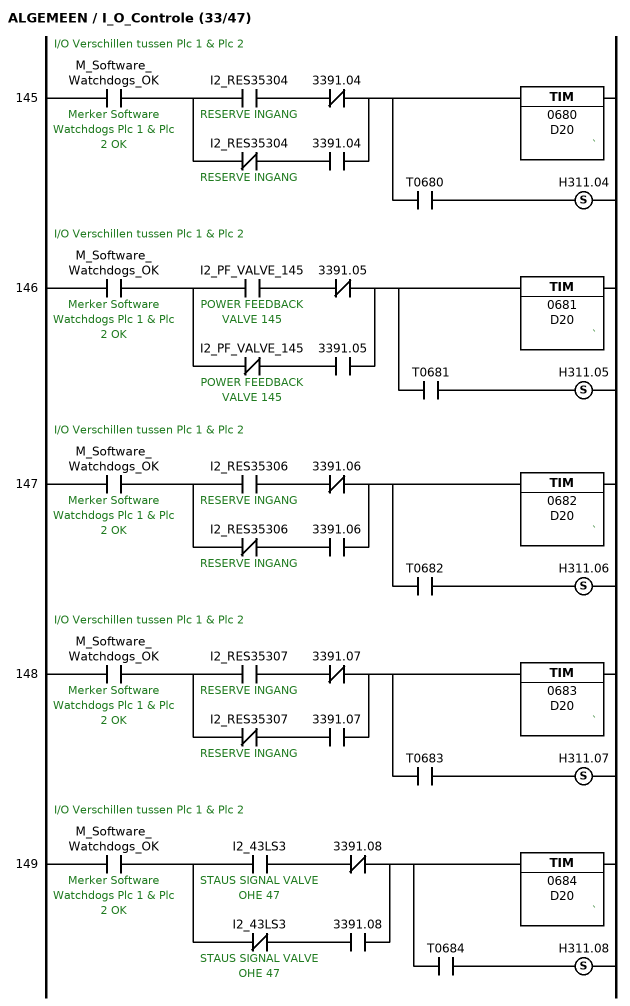
; [picture p48: ALGEMEEN / I_O_Controle, rungs 145-149]
; rung 145: I/O Verschillen tussen Plc 1 & Plc 2
LD M_Software_Watchdogs_OK  ; Merker Software Watchdogs Plc 1 & Plc 2 OK
LD I2_RES35304  ; RESERVE INGANG
ANDNOT 3391.04
LDNOT I2_RES35304  ; RESERVE INGANG
AND 3391.04
ORLD
ANDLD
TIM 0680 D20  ; `
AND T0680
SET H311.04
; rung 146: I/O Verschillen tussen Plc 1 & Plc 2
LD M_Software_Watchdogs_OK  ; Merker Software Watchdogs Plc 1 & Plc 2 OK
LD I2_PF_VALVE_145  ; POWER FEEDBACK VALVE 145
ANDNOT 3391.05
LDNOT I2_PF_VALVE_145  ; POWER FEEDBACK VALVE 145
AND 3391.05
ORLD
ANDLD
TIM 0681 D20  ; `
AND T0681
SET H311.05
; rung 147: I/O Verschillen tussen Plc 1 & Plc 2
LD M_Software_Watchdogs_OK  ; Merker Software Watchdogs Plc 1 & Plc 2 OK
LD I2_RES35306  ; RESERVE INGANG
ANDNOT 3391.06
LDNOT I2_RES35306  ; RESERVE INGANG
AND 3391.06
ORLD
ANDLD
TIM 0682 D20  ; `
AND T0682
SET H311.06
; rung 148: I/O Verschillen tussen Plc 1 & Plc 2
LD M_Software_Watchdogs_OK  ; Merker Software Watchdogs Plc 1 & Plc 2 OK
LD I2_RES35307  ; RESERVE INGANG
ANDNOT 3391.07
LDNOT I2_RES35307  ; RESERVE INGANG
AND 3391.07
ORLD
ANDLD
TIM 0683 D20  ; `
AND T0683
SET H311.07
; rung 149: I/O Verschillen tussen Plc 1 & Plc 2
LD M_Software_Watchdogs_OK  ; Merker Software Watchdogs Plc 1 & Plc 2 OK
LD I2_43LS3  ; STAUS SIGNAL VALVE OHE 47
ANDNOT 3391.08
LDNOT I2_43LS3  ; STAUS SIGNAL VALVE OHE 47
AND 3391.08
ORLD
ANDLD
TIM 0684 D20  ; `
AND T0684
SET H311.08

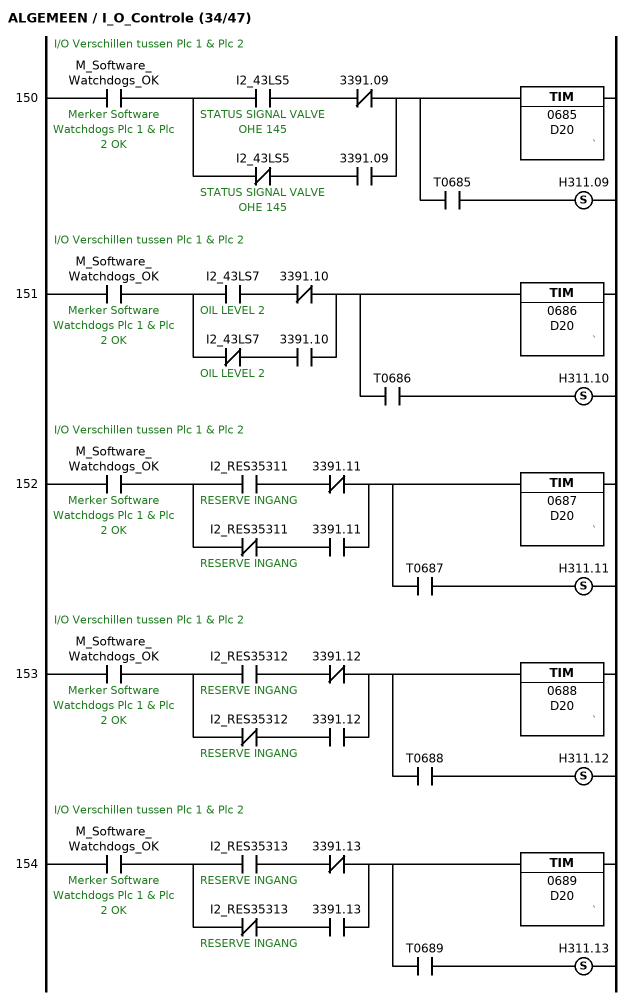
; rung 150: I/O Verschillen tussen Plc 1 & Plc 2
LD M_Software_Watchdogs_OK  ; Merker Software Watchdogs Plc 1 & Plc 2 OK
LD I2_43LS5  ; STATUS SIGNAL VALVE OHE 145
ANDNOT 3391.09
LDNOT I2_43LS5  ; STATUS SIGNAL VALVE OHE 145
AND 3391.09
ORLD
ANDLD
TIM 0685 D20  ; `
AND T0685
SET H311.09
; rung 151: I/O Verschillen tussen Plc 1 & Plc 2
LD M_Software_Watchdogs_OK  ; Merker Software Watchdogs Plc 1 & Plc 2 OK
LD I2_43LS7  ; OIL LEVEL 2
ANDNOT 3391.10
LDNOT I2_43LS7  ; OIL LEVEL 2
AND 3391.10
ORLD
ANDLD
TIM 0686 D20  ; `
AND T0686
SET H311.10
; rung 152: I/O Verschillen tussen Plc 1 & Plc 2
LD M_Software_Watchdogs_OK  ; Merker Software Watchdogs Plc 1 & Plc 2 OK
LD I2_RES35311  ; RESERVE INGANG
ANDNOT 3391.11
LDNOT I2_RES35311  ; RESERVE INGANG
AND 3391.11
ORLD
ANDLD
TIM 0687 D20  ; `
AND T0687
SET H311.11
; rung 153: I/O Verschillen tussen Plc 1 & Plc 2
LD M_Software_Watchdogs_OK  ; Merker Software Watchdogs Plc 1 & Plc 2 OK
LD I2_RES35312  ; RESERVE INGANG
ANDNOT 3391.12
LDNOT I2_RES35312  ; RESERVE INGANG
AND 3391.12
ORLD
ANDLD
TIM 0688 D20  ; `
AND T0688
SET H311.12
; rung 154: I/O Verschillen tussen Plc 1 & Plc 2
LD M_Software_Watchdogs_OK  ; Merker Software Watchdogs Plc 1 & Plc 2 OK
LD I2_RES35313  ; RESERVE INGANG
ANDNOT 3391.13
LDNOT I2_RES35313  ; RESERVE INGANG
AND 3391.13
ORLD
ANDLD
TIM 0689 D20  ; `
AND T0689
SET H311.13

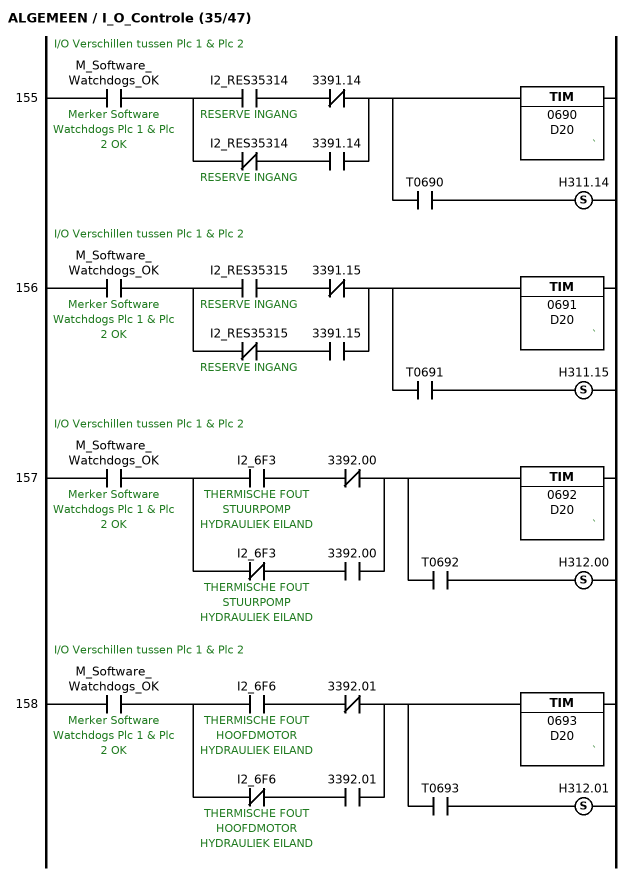
; rung 155: I/O Verschillen tussen Plc 1 & Plc 2
LD M_Software_Watchdogs_OK  ; Merker Software Watchdogs Plc 1 & Plc 2 OK
LD I2_RES35314  ; RESERVE INGANG
ANDNOT 3391.14
LDNOT I2_RES35314  ; RESERVE INGANG
AND 3391.14
ORLD
ANDLD
TIM 0690 D20  ; `
AND T0690
SET H311.14
; rung 156: I/O Verschillen tussen Plc 1 & Plc 2
LD M_Software_Watchdogs_OK  ; Merker Software Watchdogs Plc 1 & Plc 2 OK
LD I2_RES35315  ; RESERVE INGANG
ANDNOT 3391.15
LDNOT I2_RES35315  ; RESERVE INGANG
AND 3391.15
ORLD
ANDLD
TIM 0691 D20  ; `
AND T0691
SET H311.15
; rung 157: I/O Verschillen tussen Plc 1 & Plc 2
LD M_Software_Watchdogs_OK  ; Merker Software Watchdogs Plc 1 & Plc 2 OK
LD I2_6F3  ; THERMISCHE FOUT STUURPOMP HYDRAULIEK EILAND
ANDNOT 3392.00
LDNOT I2_6F3  ; THERMISCHE FOUT STUURPOMP HYDRAULIEK EILAND
AND 3392.00
ORLD
ANDLD
TIM 0692 D20  ; `
AND T0692
SET H312.00
; rung 158: I/O Verschillen tussen Plc 1 & Plc 2
LD M_Software_Watchdogs_OK  ; Merker Software Watchdogs Plc 1 & Plc 2 OK
LD I2_6F6  ; THERMISCHE FOUT HOOFDMOTOR HYDRAULIEK EILAND
ANDNOT 3392.01
LDNOT I2_6F6  ; THERMISCHE FOUT HOOFDMOTOR HYDRAULIEK EILAND
AND 3392.01
ORLD
ANDLD
TIM 0693 D20  ; `
AND T0693
SET H312.01

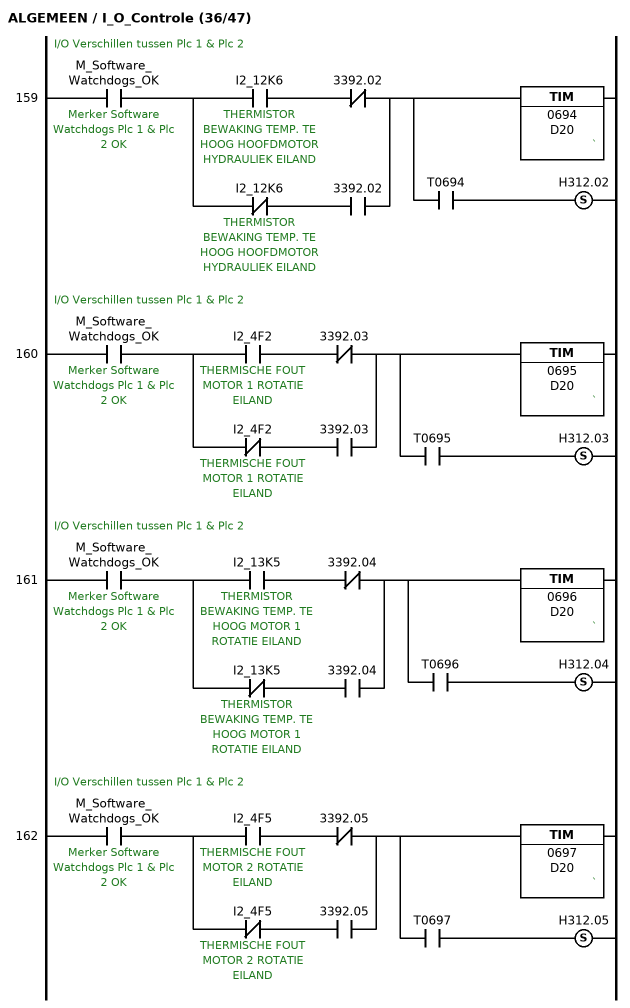
; rung 159: I/O Verschillen tussen Plc 1 & Plc 2
LD M_Software_Watchdogs_OK  ; Merker Software Watchdogs Plc 1 & Plc 2 OK
LD I2_12K6  ; THERMISTOR BEWAKING TEMP. TE HOOG HOOFDMOTOR HYDRAULIEK EILAND
ANDNOT 3392.02
LDNOT I2_12K6  ; THERMISTOR BEWAKING TEMP. TE HOOG HOOFDMOTOR HYDRAULIEK EILAND
AND 3392.02
ORLD
ANDLD
TIM 0694 D20  ; `
AND T0694
SET H312.02
; rung 160: I/O Verschillen tussen Plc 1 & Plc 2
LD M_Software_Watchdogs_OK  ; Merker Software Watchdogs Plc 1 & Plc 2 OK
LD I2_4F2  ; THERMISCHE FOUT MOTOR 1 ROTATIE EILAND
ANDNOT 3392.03
LDNOT I2_4F2  ; THERMISCHE FOUT MOTOR 1 ROTATIE EILAND
AND 3392.03
ORLD
ANDLD
TIM 0695 D20  ; `
AND T0695
SET H312.03
; rung 161: I/O Verschillen tussen Plc 1 & Plc 2
LD M_Software_Watchdogs_OK  ; Merker Software Watchdogs Plc 1 & Plc 2 OK
LD I2_13K5  ; THERMISTOR BEWAKING TEMP. TE HOOG MOTOR 1 ROTATIE EILAND
ANDNOT 3392.04
LDNOT I2_13K5  ; THERMISTOR BEWAKING TEMP. TE HOOG MOTOR 1 ROTATIE EILAND
AND 3392.04
ORLD
ANDLD
TIM 0696 D20  ; `
AND T0696
SET H312.04
; rung 162: I/O Verschillen tussen Plc 1 & Plc 2
LD M_Software_Watchdogs_OK  ; Merker Software Watchdogs Plc 1 & Plc 2 OK
LD I2_4F5  ; THERMISCHE FOUT MOTOR 2 ROTATIE EILAND
ANDNOT 3392.05
LDNOT I2_4F5  ; THERMISCHE FOUT MOTOR 2 ROTATIE EILAND
AND 3392.05
ORLD
ANDLD
TIM 0697 D20  ; `
AND T0697
SET H312.05

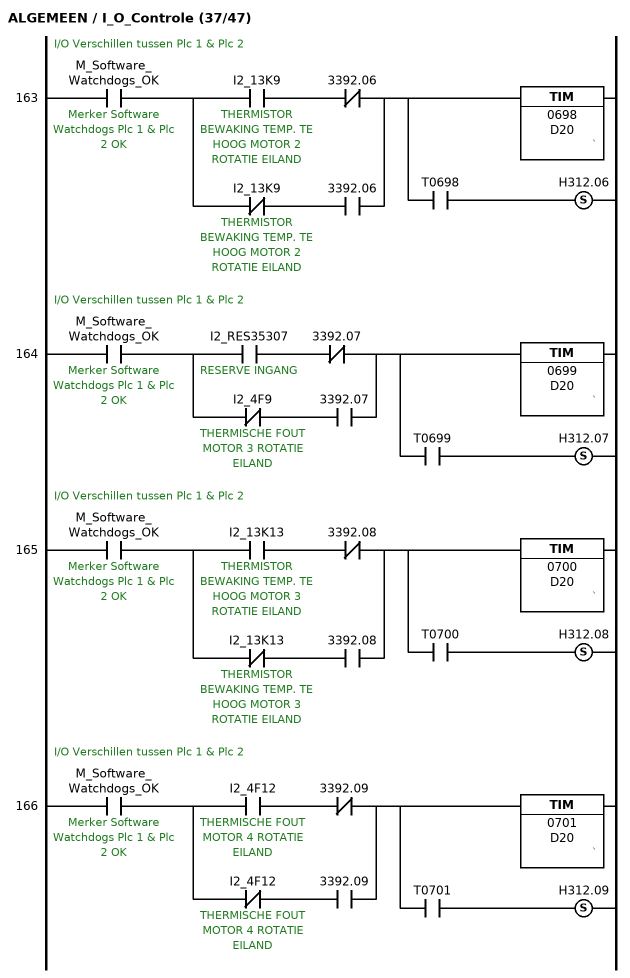
; rung 163: I/O Verschillen tussen Plc 1 & Plc 2
LD M_Software_Watchdogs_OK  ; Merker Software Watchdogs Plc 1 & Plc 2 OK
LD I2_13K9  ; THERMISTOR BEWAKING TEMP. TE HOOG MOTOR 2 ROTATIE EILAND
ANDNOT 3392.06
LDNOT I2_13K9  ; THERMISTOR BEWAKING TEMP. TE HOOG MOTOR 2 ROTATIE EILAND
AND 3392.06
ORLD
ANDLD
TIM 0698 D20  ; `
AND T0698
SET H312.06
; rung 164: I/O Verschillen tussen Plc 1 & Plc 2
LD M_Software_Watchdogs_OK  ; Merker Software Watchdogs Plc 1 & Plc 2 OK
LD I2_RES35307  ; RESERVE INGANG
ANDNOT 3392.07
LDNOT I2_4F9  ; THERMISCHE FOUT MOTOR 3 ROTATIE EILAND
AND 3392.07
ORLD
ANDLD
TIM 0699 D20  ; `
AND T0699
SET H312.07
; rung 165: I/O Verschillen tussen Plc 1 & Plc 2
LD M_Software_Watchdogs_OK  ; Merker Software Watchdogs Plc 1 & Plc 2 OK
LD I2_13K13  ; THERMISTOR BEWAKING TEMP. TE HOOG MOTOR 3 ROTATIE EILAND
ANDNOT 3392.08
LDNOT I2_13K13  ; THERMISTOR BEWAKING TEMP. TE HOOG MOTOR 3 ROTATIE EILAND
AND 3392.08
ORLD
ANDLD
TIM 0700 D20  ; `
AND T0700
SET H312.08
; rung 166: I/O Verschillen tussen Plc 1 & Plc 2
LD M_Software_Watchdogs_OK  ; Merker Software Watchdogs Plc 1 & Plc 2 OK
LD I2_4F12  ; THERMISCHE FOUT MOTOR 4 ROTATIE EILAND
ANDNOT 3392.09
LDNOT I2_4F12  ; THERMISCHE FOUT MOTOR 4 ROTATIE EILAND
AND 3392.09
ORLD
ANDLD
TIM 0701 D20  ; `
AND T0701
SET H312.09

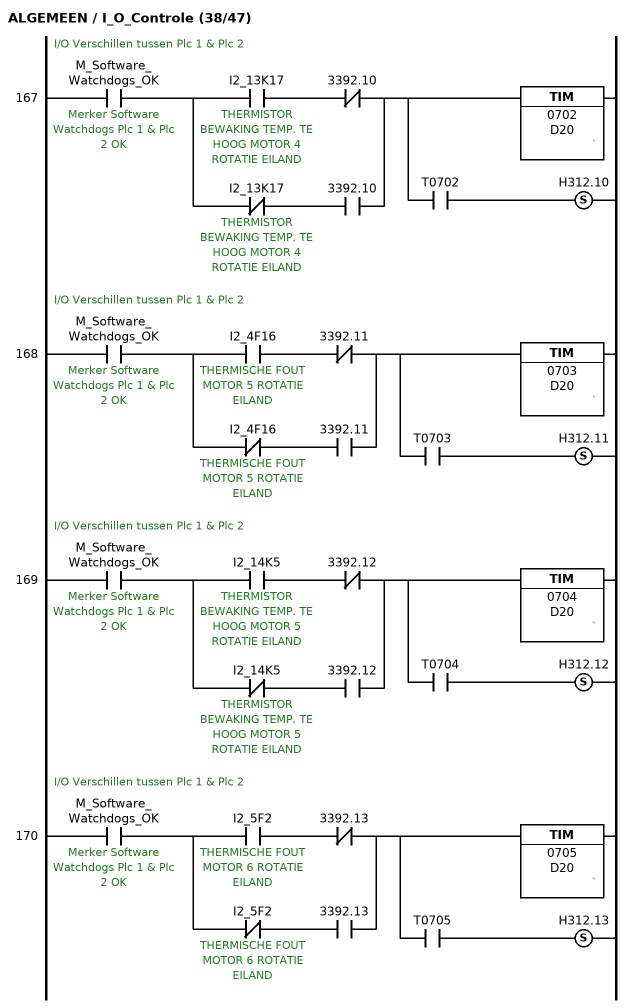
; rung 167: I/O Verschillen tussen Plc 1 & Plc 2
LD M_Software_Watchdogs_OK  ; Merker Software Watchdogs Plc 1 & Plc 2 OK
LD I2_13K17  ; THERMISTOR BEWAKING TEMP. TE HOOG MOTOR 4 ROTATIE EILAND
ANDNOT 3392.10
LDNOT I2_13K17  ; THERMISTOR BEWAKING TEMP. TE HOOG MOTOR 4 ROTATIE EILAND
AND 3392.10
ORLD
ANDLD
TIM 0702 D20  ; `
AND T0702
SET H312.10
; rung 168: I/O Verschillen tussen Plc 1 & Plc 2
LD M_Software_Watchdogs_OK  ; Merker Software Watchdogs Plc 1 & Plc 2 OK
LD I2_4F16  ; THERMISCHE FOUT MOTOR 5 ROTATIE EILAND
ANDNOT 3392.11
LDNOT I2_4F16  ; THERMISCHE FOUT MOTOR 5 ROTATIE EILAND
AND 3392.11
ORLD
ANDLD
TIM 0703 D20  ; `
AND T0703
SET H312.11
; rung 169: I/O Verschillen tussen Plc 1 & Plc 2
LD M_Software_Watchdogs_OK  ; Merker Software Watchdogs Plc 1 & Plc 2 OK
LD I2_14K5  ; THERMISTOR BEWAKING TEMP. TE HOOG MOTOR 5 ROTATIE EILAND
ANDNOT 3392.12
LDNOT I2_14K5  ; THERMISTOR BEWAKING TEMP. TE HOOG MOTOR 5 ROTATIE EILAND
AND 3392.12
ORLD
ANDLD
TIM 0704 D20  ; `
AND T0704
SET H312.12
; rung 170: I/O Verschillen tussen Plc 1 & Plc 2
LD M_Software_Watchdogs_OK  ; Merker Software Watchdogs Plc 1 & Plc 2 OK
LD I2_5F2  ; THERMISCHE FOUT MOTOR 6 ROTATIE EILAND
ANDNOT 3392.13
LDNOT I2_5F2  ; THERMISCHE FOUT MOTOR 6 ROTATIE EILAND
AND 3392.13
ORLD
ANDLD
TIM 0705 D20  ; `
AND T0705
SET H312.13

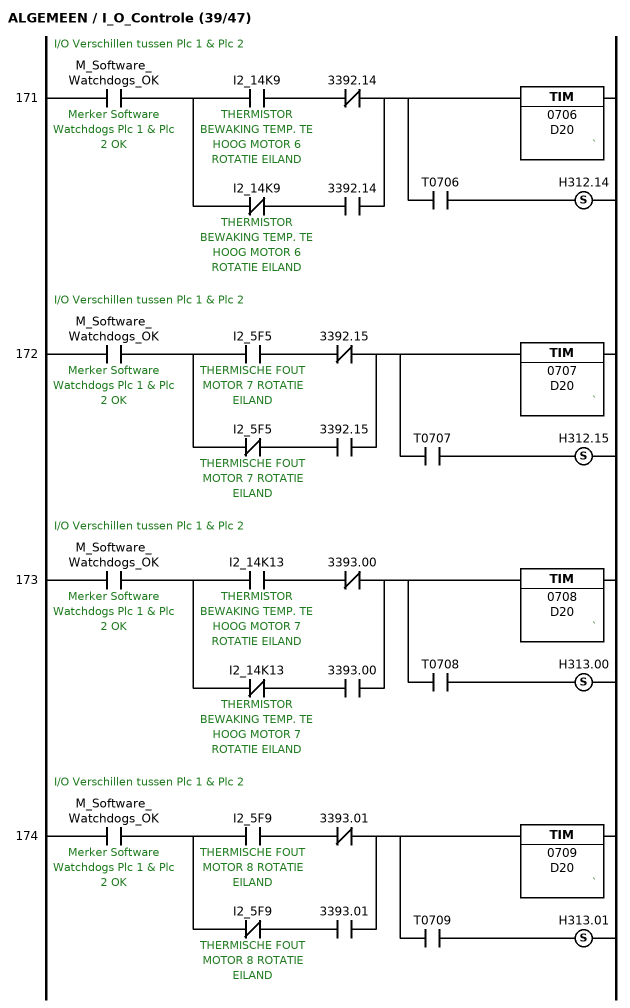
; rung 171: I/O Verschillen tussen Plc 1 & Plc 2
LD M_Software_Watchdogs_OK  ; Merker Software Watchdogs Plc 1 & Plc 2 OK
LD I2_14K9  ; THERMISTOR BEWAKING TEMP. TE HOOG MOTOR 6 ROTATIE EILAND
ANDNOT 3392.14
LDNOT I2_14K9  ; THERMISTOR BEWAKING TEMP. TE HOOG MOTOR 6 ROTATIE EILAND
AND 3392.14
ORLD
ANDLD
TIM 0706 D20  ; `
AND T0706
SET H312.14
; rung 172: I/O Verschillen tussen Plc 1 & Plc 2
LD M_Software_Watchdogs_OK  ; Merker Software Watchdogs Plc 1 & Plc 2 OK
LD I2_5F5  ; THERMISCHE FOUT MOTOR 7 ROTATIE EILAND
ANDNOT 3392.15
LDNOT I2_5F5  ; THERMISCHE FOUT MOTOR 7 ROTATIE EILAND
AND 3392.15
ORLD
ANDLD
TIM 0707 D20  ; `
AND T0707
SET H312.15
; rung 173: I/O Verschillen tussen Plc 1 & Plc 2
LD M_Software_Watchdogs_OK  ; Merker Software Watchdogs Plc 1 & Plc 2 OK
LD I2_14K13  ; THERMISTOR BEWAKING TEMP. TE HOOG MOTOR 7 ROTATIE EILAND
ANDNOT 3393.00
LDNOT I2_14K13  ; THERMISTOR BEWAKING TEMP. TE HOOG MOTOR 7 ROTATIE EILAND
AND 3393.00
ORLD
ANDLD
TIM 0708 D20  ; `
AND T0708
SET H313.00
; rung 174: I/O Verschillen tussen Plc 1 & Plc 2
LD M_Software_Watchdogs_OK  ; Merker Software Watchdogs Plc 1 & Plc 2 OK
LD I2_5F9  ; THERMISCHE FOUT MOTOR 8 ROTATIE EILAND
ANDNOT 3393.01
LDNOT I2_5F9  ; THERMISCHE FOUT MOTOR 8 ROTATIE EILAND
AND 3393.01
ORLD
ANDLD
TIM 0709 D20  ; `
AND T0709
SET H313.01

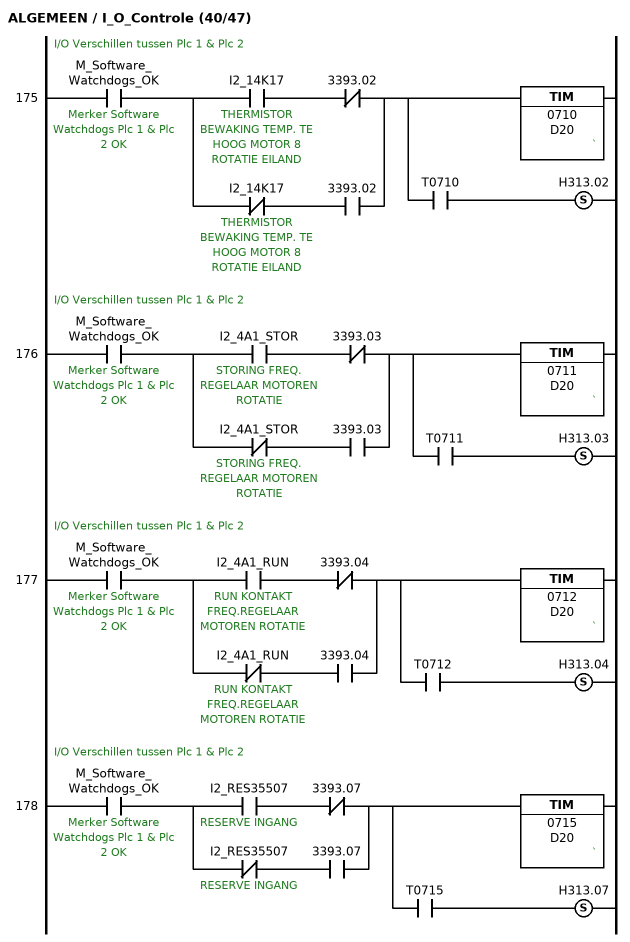
; rung 175: I/O Verschillen tussen Plc 1 & Plc 2
LD M_Software_Watchdogs_OK  ; Merker Software Watchdogs Plc 1 & Plc 2 OK
LD I2_14K17  ; THERMISTOR BEWAKING TEMP. TE HOOG MOTOR 8 ROTATIE EILAND
ANDNOT 3393.02
LDNOT I2_14K17  ; THERMISTOR BEWAKING TEMP. TE HOOG MOTOR 8 ROTATIE EILAND
AND 3393.02
ORLD
ANDLD
TIM 0710 D20  ; `
AND T0710
SET H313.02
; rung 176: I/O Verschillen tussen Plc 1 & Plc 2
LD M_Software_Watchdogs_OK  ; Merker Software Watchdogs Plc 1 & Plc 2 OK
LD I2_4A1_STOR  ; STORING FREQ.REGELAAR MOTOREN ROTATIE
ANDNOT 3393.03
LDNOT I2_4A1_STOR  ; STORING FREQ.REGELAAR MOTOREN ROTATIE
AND 3393.03
ORLD
ANDLD
TIM 0711 D20  ; `
AND T0711
SET H313.03
; rung 177: I/O Verschillen tussen Plc 1 & Plc 2
LD M_Software_Watchdogs_OK  ; Merker Software Watchdogs Plc 1 & Plc 2 OK
LD I2_4A1_RUN  ; RUN KONTAKT FREQ.REGELAAR MOTOREN ROTATIE
ANDNOT 3393.04
LDNOT I2_4A1_RUN  ; RUN KONTAKT FREQ.REGELAAR MOTOREN ROTATIE
AND 3393.04
ORLD
ANDLD
TIM 0712 D20  ; `
AND T0712
SET H313.04
; rung 178: I/O Verschillen tussen Plc 1 & Plc 2
LD M_Software_Watchdogs_OK  ; Merker Software Watchdogs Plc 1 & Plc 2 OK
LD I2_RES35507  ; RESERVE INGANG
ANDNOT 3393.07
LDNOT I2_RES35507  ; RESERVE INGANG
AND 3393.07
ORLD
ANDLD
TIM 0715 D20  ; `
AND T0715
SET H313.07

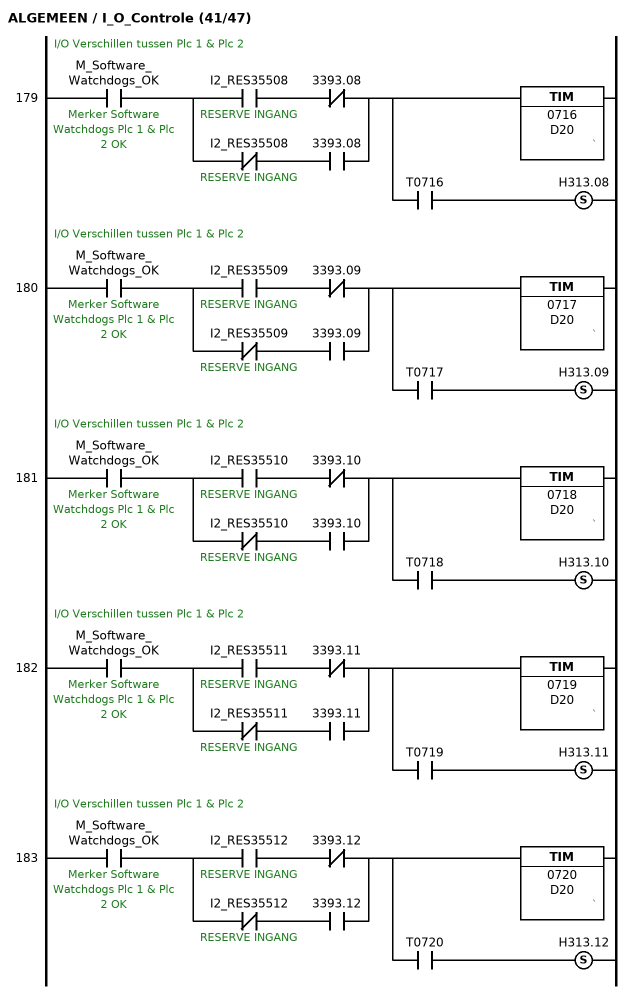
; rung 179: I/O Verschillen tussen Plc 1 & Plc 2
LD M_Software_Watchdogs_OK  ; Merker Software Watchdogs Plc 1 & Plc 2 OK
LD I2_RES35508  ; RESERVE INGANG
ANDNOT 3393.08
LDNOT I2_RES35508  ; RESERVE INGANG
AND 3393.08
ORLD
ANDLD
TIM 0716 D20  ; `
AND T0716
SET H313.08
; rung 180: I/O Verschillen tussen Plc 1 & Plc 2
LD M_Software_Watchdogs_OK  ; Merker Software Watchdogs Plc 1 & Plc 2 OK
LD I2_RES35509  ; RESERVE INGANG
ANDNOT 3393.09
LDNOT I2_RES35509  ; RESERVE INGANG
AND 3393.09
ORLD
ANDLD
TIM 0717 D20  ; `
AND T0717
SET H313.09
; rung 181: I/O Verschillen tussen Plc 1 & Plc 2
LD M_Software_Watchdogs_OK  ; Merker Software Watchdogs Plc 1 & Plc 2 OK
LD I2_RES35510  ; RESERVE INGANG
ANDNOT 3393.10
LDNOT I2_RES35510  ; RESERVE INGANG
AND 3393.10
ORLD
ANDLD
TIM 0718 D20  ; `
AND T0718
SET H313.10
; rung 182: I/O Verschillen tussen Plc 1 & Plc 2
LD M_Software_Watchdogs_OK  ; Merker Software Watchdogs Plc 1 & Plc 2 OK
LD I2_RES35511  ; RESERVE INGANG
ANDNOT 3393.11
LDNOT I2_RES35511  ; RESERVE INGANG
AND 3393.11
ORLD
ANDLD
TIM 0719 D20  ; `
AND T0719
SET H313.11
; rung 183: I/O Verschillen tussen Plc 1 & Plc 2
LD M_Software_Watchdogs_OK  ; Merker Software Watchdogs Plc 1 & Plc 2 OK
LD I2_RES35512  ; RESERVE INGANG
ANDNOT 3393.12
LDNOT I2_RES35512  ; RESERVE INGANG
AND 3393.12
ORLD
ANDLD
TIM 0720 D20  ; `
AND T0720
SET H313.12

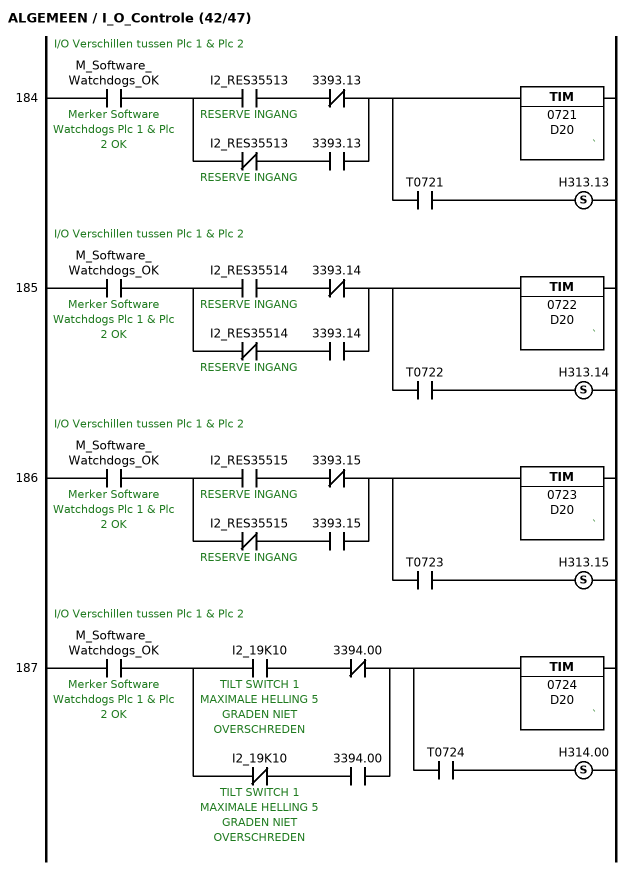
; rung 184: I/O Verschillen tussen Plc 1 & Plc 2
LD M_Software_Watchdogs_OK  ; Merker Software Watchdogs Plc 1 & Plc 2 OK
LD I2_RES35513  ; RESERVE INGANG
ANDNOT 3393.13
LDNOT I2_RES35513  ; RESERVE INGANG
AND 3393.13
ORLD
ANDLD
TIM 0721 D20  ; `
AND T0721
SET H313.13
; rung 185: I/O Verschillen tussen Plc 1 & Plc 2
LD M_Software_Watchdogs_OK  ; Merker Software Watchdogs Plc 1 & Plc 2 OK
LD I2_RES35514  ; RESERVE INGANG
ANDNOT 3393.14
LDNOT I2_RES35514  ; RESERVE INGANG
AND 3393.14
ORLD
ANDLD
TIM 0722 D20  ; `
AND T0722
SET H313.14
; rung 186: I/O Verschillen tussen Plc 1 & Plc 2
LD M_Software_Watchdogs_OK  ; Merker Software Watchdogs Plc 1 & Plc 2 OK
LD I2_RES35515  ; RESERVE INGANG
ANDNOT 3393.15
LDNOT I2_RES35515  ; RESERVE INGANG
AND 3393.15
ORLD
ANDLD
TIM 0723 D20  ; `
AND T0723
SET H313.15
; rung 187: I/O Verschillen tussen Plc 1 & Plc 2
LD M_Software_Watchdogs_OK  ; Merker Software Watchdogs Plc 1 & Plc 2 OK
LD I2_19K10  ; TILT SWITCH 1 MAXIMALE HELLING 5 GRADEN NIET OVERSCHREDEN
ANDNOT 3394.00
LDNOT I2_19K10  ; TILT SWITCH 1 MAXIMALE HELLING 5 GRADEN NIET OVERSCHREDEN
AND 3394.00
ORLD
ANDLD
TIM 0724 D20  ; `
AND T0724
SET H314.00

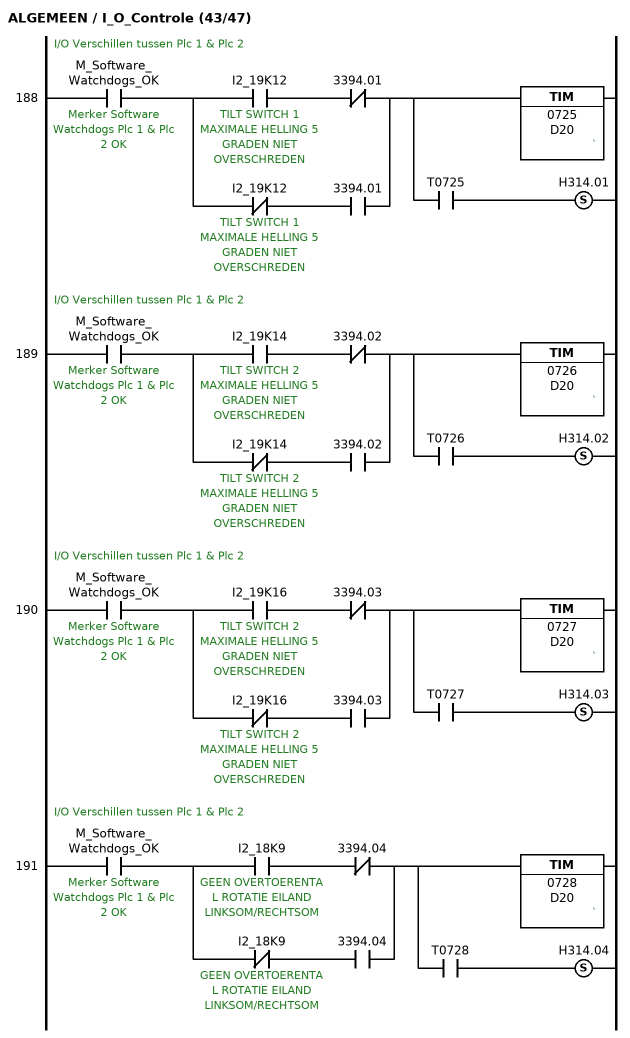
; rung 188: I/O Verschillen tussen Plc 1 & Plc 2
LD M_Software_Watchdogs_OK  ; Merker Software Watchdogs Plc 1 & Plc 2 OK
LD I2_19K12  ; TILT SWITCH 1 MAXIMALE HELLING 5 GRADEN NIET OVERSCHREDEN
ANDNOT 3394.01
LDNOT I2_19K12  ; TILT SWITCH 1 MAXIMALE HELLING 5 GRADEN NIET OVERSCHREDEN
AND 3394.01
ORLD
ANDLD
TIM 0725 D20  ; `
AND T0725
SET H314.01
; rung 189: I/O Verschillen tussen Plc 1 & Plc 2
LD M_Software_Watchdogs_OK  ; Merker Software Watchdogs Plc 1 & Plc 2 OK
LD I2_19K14  ; TILT SWITCH 2 MAXIMALE HELLING 5 GRADEN NIET OVERSCHREDEN
ANDNOT 3394.02
LDNOT I2_19K14  ; TILT SWITCH 2 MAXIMALE HELLING 5 GRADEN NIET OVERSCHREDEN
AND 3394.02
ORLD
ANDLD
TIM 0726 D20  ; `
AND T0726
SET H314.02
; rung 190: I/O Verschillen tussen Plc 1 & Plc 2
LD M_Software_Watchdogs_OK  ; Merker Software Watchdogs Plc 1 & Plc 2 OK
LD I2_19K16  ; TILT SWITCH 2 MAXIMALE HELLING 5 GRADEN NIET OVERSCHREDEN
ANDNOT 3394.03
LDNOT I2_19K16  ; TILT SWITCH 2 MAXIMALE HELLING 5 GRADEN NIET OVERSCHREDEN
AND 3394.03
ORLD
ANDLD
TIM 0727 D20  ; `
AND T0727
SET H314.03
; rung 191: I/O Verschillen tussen Plc 1 & Plc 2
LD M_Software_Watchdogs_OK  ; Merker Software Watchdogs Plc 1 & Plc 2 OK
LD I2_18K9  ; GEEN OVERTOERENTAL ROTATIE EILAND LINKSOM/RECHTSOM
ANDNOT 3394.04
LDNOT I2_18K9  ; GEEN OVERTOERENTAL ROTATIE EILAND LINKSOM/RECHTSOM
AND 3394.04
ORLD
ANDLD
TIM 0728 D20  ; `
AND T0728
SET H314.04

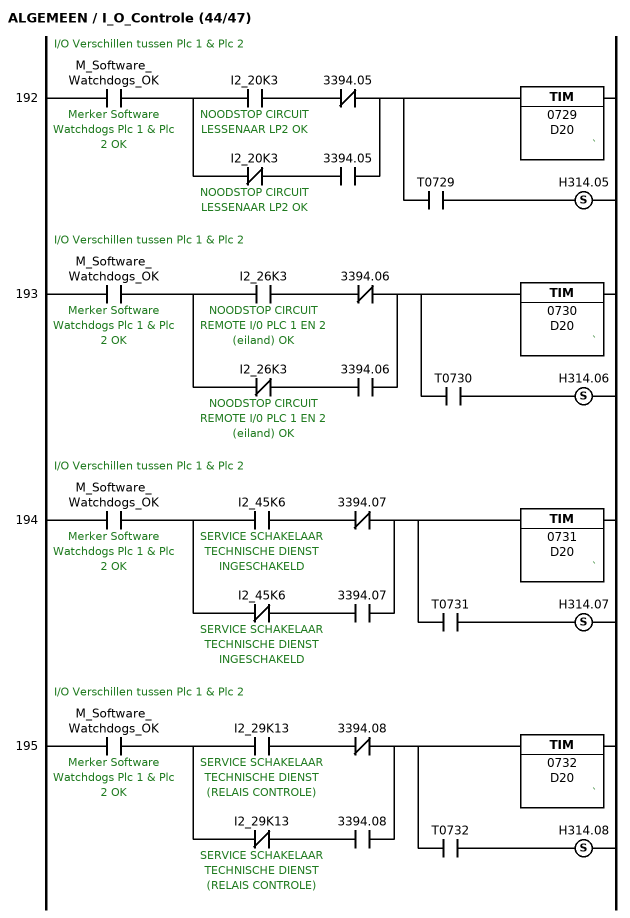
; rung 192: I/O Verschillen tussen Plc 1 & Plc 2
LD M_Software_Watchdogs_OK  ; Merker Software Watchdogs Plc 1 & Plc 2 OK
LD I2_20K3  ; NOODSTOP CIRCUIT LESSENAAR LP2 OK
ANDNOT 3394.05
LDNOT I2_20K3  ; NOODSTOP CIRCUIT LESSENAAR LP2 OK
AND 3394.05
ORLD
ANDLD
TIM 0729 D20  ; `
AND T0729
SET H314.05
; rung 193: I/O Verschillen tussen Plc 1 & Plc 2
LD M_Software_Watchdogs_OK  ; Merker Software Watchdogs Plc 1 & Plc 2 OK
LD I2_26K3  ; NOODSTOP CIRCUIT REMOTE I/0 PLC 1 EN 2 (eiland) OK
ANDNOT 3394.06
LDNOT I2_26K3  ; NOODSTOP CIRCUIT REMOTE I/0 PLC 1 EN 2 (eiland) OK
AND 3394.06
ORLD
ANDLD
TIM 0730 D20  ; `
AND T0730
SET H314.06
; rung 194: I/O Verschillen tussen Plc 1 & Plc 2
LD M_Software_Watchdogs_OK  ; Merker Software Watchdogs Plc 1 & Plc 2 OK
LD I2_45K6  ; SERVICE SCHAKELAAR TECHNISCHE DIENST INGESCHAKELD
ANDNOT 3394.07
LDNOT I2_45K6  ; SERVICE SCHAKELAAR TECHNISCHE DIENST INGESCHAKELD
AND 3394.07
ORLD
ANDLD
TIM 0731 D20  ; `
AND T0731
SET H314.07
; rung 195: I/O Verschillen tussen Plc 1 & Plc 2
LD M_Software_Watchdogs_OK  ; Merker Software Watchdogs Plc 1 & Plc 2 OK
LD I2_29K13  ; SERVICE SCHAKELAAR TECHNISCHE DIENST (RELAIS CONTROLE)
ANDNOT 3394.08
LDNOT I2_29K13  ; SERVICE SCHAKELAAR TECHNISCHE DIENST (RELAIS CONTROLE)
AND 3394.08
ORLD
ANDLD
TIM 0732 D20  ; `
AND T0732
SET H314.08

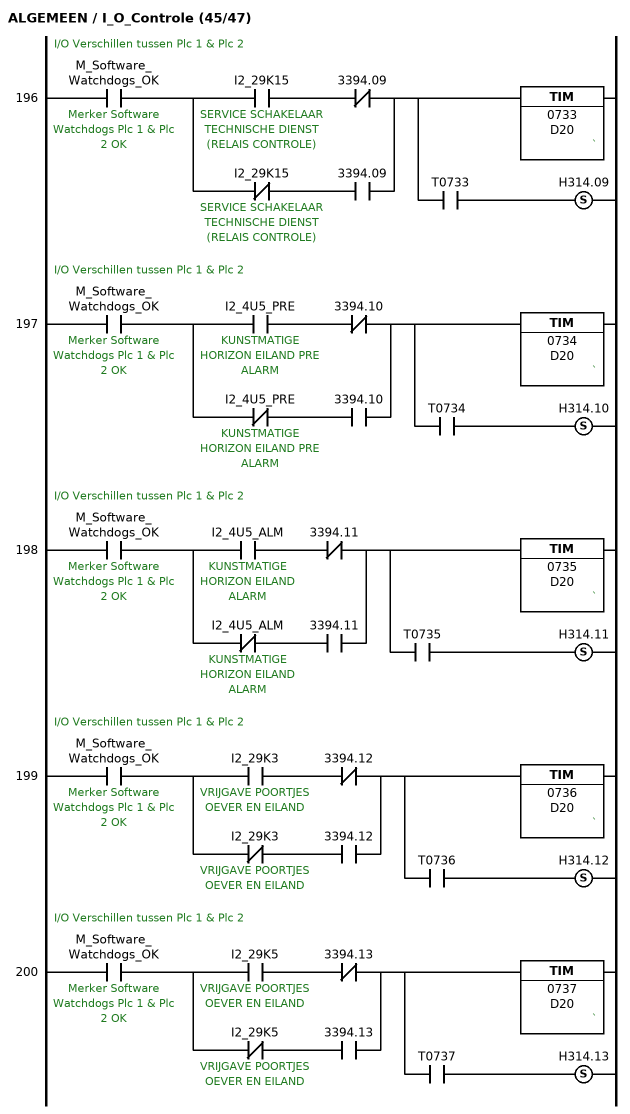
; rung 196: I/O Verschillen tussen Plc 1 & Plc 2
LD M_Software_Watchdogs_OK  ; Merker Software Watchdogs Plc 1 & Plc 2 OK
LD I2_29K15  ; SERVICE SCHAKELAAR TECHNISCHE DIENST (RELAIS CONTROLE)
ANDNOT 3394.09
LDNOT I2_29K15  ; SERVICE SCHAKELAAR TECHNISCHE DIENST (RELAIS CONTROLE)
AND 3394.09
ORLD
ANDLD
TIM 0733 D20  ; `
AND T0733
SET H314.09
; rung 197: I/O Verschillen tussen Plc 1 & Plc 2
LD M_Software_Watchdogs_OK  ; Merker Software Watchdogs Plc 1 & Plc 2 OK
LD I2_4U5_PRE  ; KUNSTMATIGE HORIZON EILAND PRE ALARM
ANDNOT 3394.10
LDNOT I2_4U5_PRE  ; KUNSTMATIGE HORIZON EILAND PRE ALARM
AND 3394.10
ORLD
ANDLD
TIM 0734 D20  ; `
AND T0734
SET H314.10
; rung 198: I/O Verschillen tussen Plc 1 & Plc 2
LD M_Software_Watchdogs_OK  ; Merker Software Watchdogs Plc 1 & Plc 2 OK
LD I2_4U5_ALM  ; KUNSTMATIGE HORIZON EILAND ALARM
ANDNOT 3394.11
LDNOT I2_4U5_ALM  ; KUNSTMATIGE HORIZON EILAND ALARM
AND 3394.11
ORLD
ANDLD
TIM 0735 D20  ; `
AND T0735
SET H314.11
; rung 199: I/O Verschillen tussen Plc 1 & Plc 2
LD M_Software_Watchdogs_OK  ; Merker Software Watchdogs Plc 1 & Plc 2 OK
LD I2_29K3  ; VRIJGAVE POORTJES OEVER EN EILAND
ANDNOT 3394.12
LDNOT I2_29K3  ; VRIJGAVE POORTJES OEVER EN EILAND
AND 3394.12
ORLD
ANDLD
TIM 0736 D20  ; `
AND T0736
SET H314.12
; rung 200: I/O Verschillen tussen Plc 1 & Plc 2
LD M_Software_Watchdogs_OK  ; Merker Software Watchdogs Plc 1 & Plc 2 OK
LD I2_29K5  ; VRIJGAVE POORTJES OEVER EN EILAND
ANDNOT 3394.13
LDNOT I2_29K5  ; VRIJGAVE POORTJES OEVER EN EILAND
AND 3394.13
ORLD
ANDLD
TIM 0737 D20  ; `
AND T0737
SET H314.13

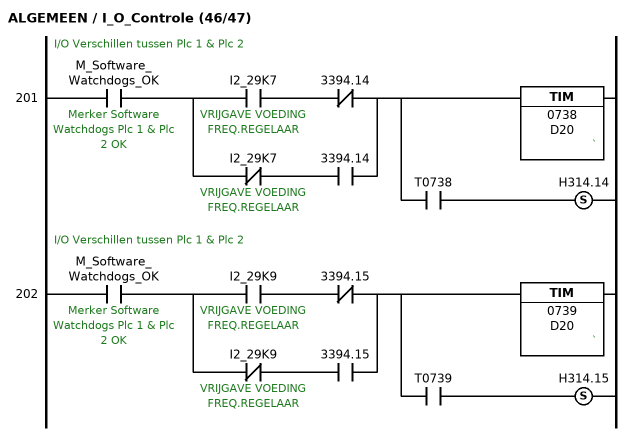
; rung 201: I/O Verschillen tussen Plc 1 & Plc 2
LD M_Software_Watchdogs_OK  ; Merker Software Watchdogs Plc 1 & Plc 2 OK
LD I2_29K7  ; VRIJGAVE VOEDING FREQ.REGELAAR
ANDNOT 3394.14
LDNOT I2_29K7  ; VRIJGAVE VOEDING FREQ.REGELAAR
AND 3394.14
ORLD
ANDLD
TIM 0738 D20  ; `
AND T0738
SET H314.14
; rung 202: I/O Verschillen tussen Plc 1 & Plc 2
LD M_Software_Watchdogs_OK  ; Merker Software Watchdogs Plc 1 & Plc 2 OK
LD I2_29K9  ; VRIJGAVE VOEDING FREQ.REGELAAR
ANDNOT 3394.15
LDNOT I2_29K9  ; VRIJGAVE VOEDING FREQ.REGELAAR
AND 3394.15
ORLD
ANDLD
TIM 0739 D20  ; `
AND T0739
SET H314.15

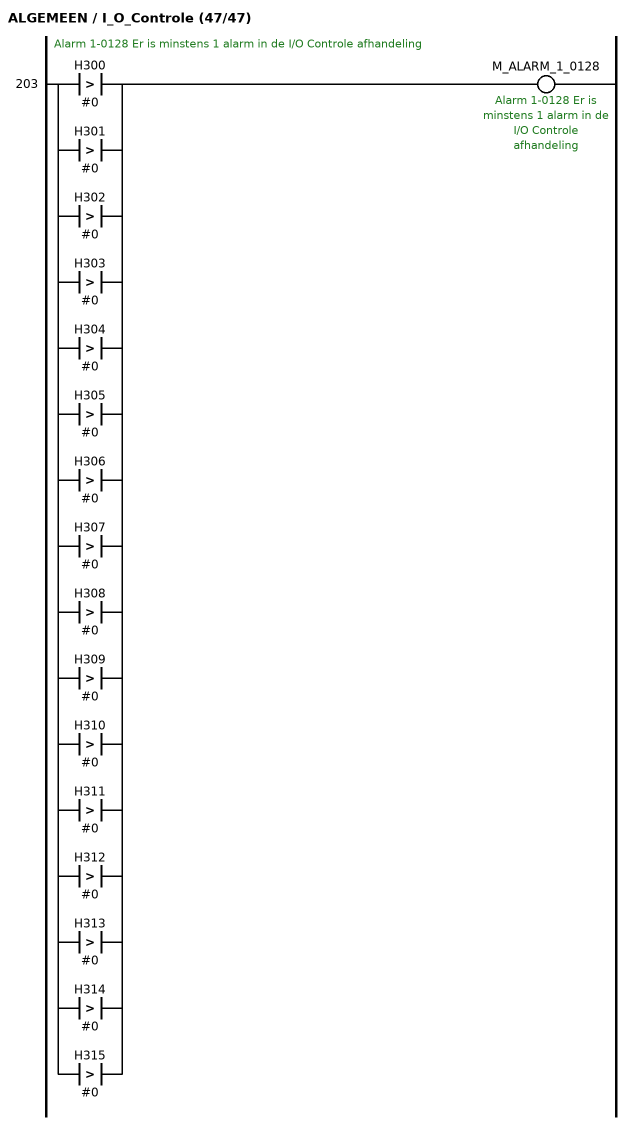
; rung 203: Alarm 1-0128 Er is minstens 1 alarm in de I/O Controle afhandeling
LD>(320) H300 #0
OR>(320) H301 #0
OR>(320) H302 #0
OR>(320) H303 #0
OR>(320) H304 #0
OR>(320) H305 #0
OR>(320) H306 #0
OR>(320) H307 #0
OR>(320) H308 #0
OR>(320) H309 #0
OR>(320) H310 #0
OR>(320) H311 #0
OR>(320) H312 #0
OR>(320) H313 #0
OR>(320) H314 #0
OR>(320) H315 #0
OUT M_ALARM_1_0128  ; Alarm 1-0128 Er is minstens 1 alarm in de I/O Controle afhandeling

### Section Watch_Dog

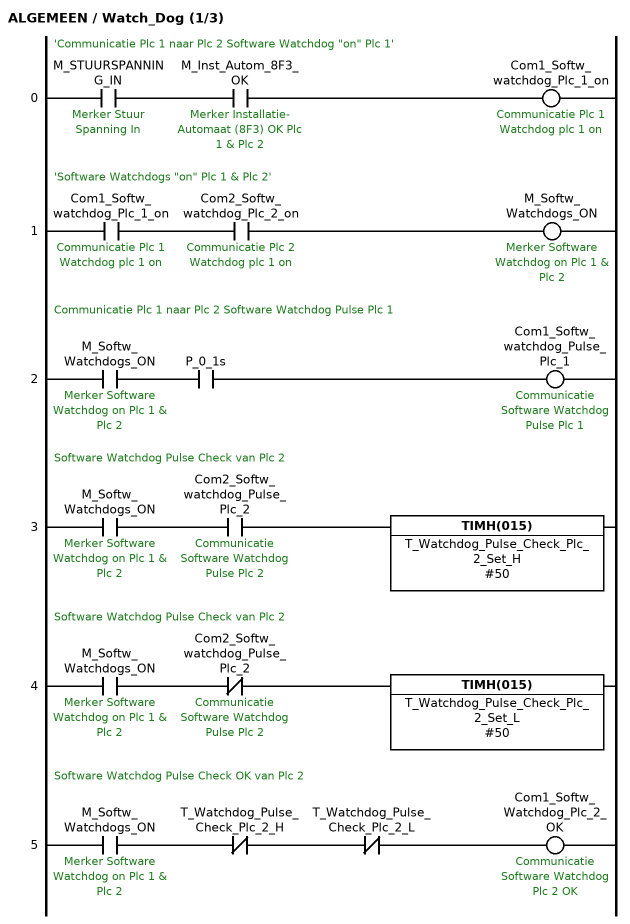
; rung 0: 'Communicatie Plc 1 naar Plc 2 Software Watchdog "on" Plc 1'
LD M_STUURSPANNING_IN  ; Merker Stuur Spanning In
AND M_Inst_Autom_8F3_OK  ; Merker Installatie-Automaat (8F3) OK Plc 1 & Plc 2
OUT Com1_Softw_watchdog_Plc_1_on  ; Communicatie Plc 1 Watchdog plc 1 on
; rung 1: 'Software Watchdogs "on" Plc 1 & Plc 2'
LD Com1_Softw_watchdog_Plc_1_on  ; Communicatie Plc 1 Watchdog plc 1 on
AND Com2_Softw_watchdog_Plc_2_on  ; Communicatie Plc 2 Watchdog plc 1 on
OUT M_Softw_Watchdogs_ON  ; Merker Software Watchdog on Plc 1 & Plc 2
; rung 2: Communicatie Plc 1 naar Plc 2 Software Watchdog Pulse Plc 1
LD M_Softw_Watchdogs_ON  ; Merker Software Watchdog on Plc 1 & Plc 2
AND P_0_1s
OUT Com1_Softw_watchdog_Pulse_Plc_1  ; Communicatie Software Watchdog Pulse Plc 1
; rung 3: Software Watchdog Pulse Check van Plc 2
LD M_Softw_Watchdogs_ON  ; Merker Software Watchdog on Plc 1 & Plc 2
AND Com2_Softw_watchdog_Pulse_Plc_2  ; Communicatie Software Watchdog Pulse Plc 2
TIMH(015) T_Watchdog_Pulse_Check_Plc_2_Set_H #50
; rung 4: Software Watchdog Pulse Check van Plc 2
LD M_Softw_Watchdogs_ON  ; Merker Software Watchdog on Plc 1 & Plc 2
ANDNOT Com2_Softw_watchdog_Pulse_Plc_2  ; Communicatie Software Watchdog Pulse Plc 2
TIMH(015) T_Watchdog_Pulse_Check_Plc_2_Set_L #50
; rung 5: Software Watchdog Pulse Check OK van Plc 2
LD M_Softw_Watchdogs_ON  ; Merker Software Watchdog on Plc 1 & Plc 2
ANDNOT T_Watchdog_Pulse_Check_Plc_2_H
ANDNOT T_Watchdog_Pulse_Check_Plc_2_L
OUT Com1_Softw_Watchdog_Plc_2_OK  ; Communicatie Software Watchdog Plc 2 OK

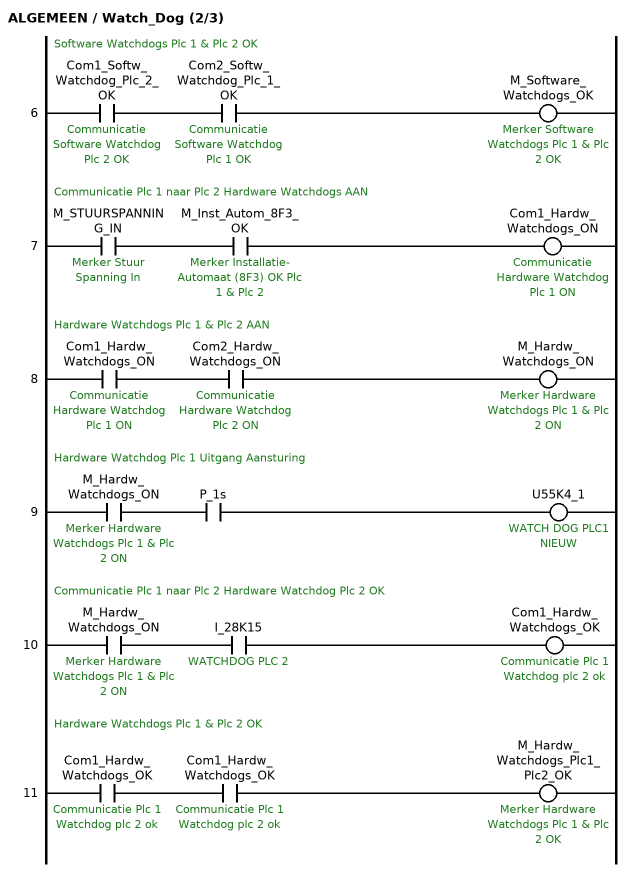
; rung 6: Software Watchdogs Plc 1 & Plc 2 OK
LD Com1_Softw_Watchdog_Plc_2_OK  ; Communicatie Software Watchdog Plc 2 OK
AND Com2_Softw_Watchdog_Plc_1_OK  ; Communicatie Software Watchdog Plc 1 OK
OUT M_Software_Watchdogs_OK  ; Merker Software Watchdogs Plc 1 & Plc 2 OK
; rung 7: Communicatie Plc 1 naar Plc 2 Hardware Watchdogs AAN
LD M_STUURSPANNING_IN  ; Merker Stuur Spanning In
AND M_Inst_Autom_8F3_OK  ; Merker Installatie-Automaat (8F3) OK Plc 1 & Plc 2
OUT Com1_Hardw_Watchdogs_ON  ; Communicatie Hardware Watchdog Plc 1 ON
; rung 8: Hardware Watchdogs Plc 1 & Plc 2 AAN
LD Com1_Hardw_Watchdogs_ON  ; Communicatie Hardware Watchdog Plc 1 ON
AND Com2_Hardw_Watchdogs_ON  ; Communicatie Hardware Watchdog Plc 2 ON
OUT M_Hardw_Watchdogs_ON  ; Merker Hardware Watchdogs Plc 1 & Plc 2 ON
; rung 9: Hardware Watchdog Plc 1 Uitgang Aansturing
LD M_Hardw_Watchdogs_ON  ; Merker Hardware Watchdogs Plc 1 & Plc 2 ON
AND P_1s
OUT U55K4_1  ; WATCH DOG PLC1 NIEUW
; rung 10: Communicatie Plc 1 naar Plc 2 Hardware Watchdog Plc 2 OK
LD M_Hardw_Watchdogs_ON  ; Merker Hardware Watchdogs Plc 1 & Plc 2 ON
AND I_28K15  ; WATCHDOG PLC 2
OUT Com1_Hardw_Watchdogs_OK  ; Communicatie Plc 1 Watchdog plc 2 ok
; rung 11: Hardware Watchdogs Plc 1 & Plc 2 OK
LD Com1_Hardw_Watchdogs_OK  ; Communicatie Plc 1 Watchdog plc 2 ok
AND Com1_Hardw_Watchdogs_OK  ; Communicatie Plc 1 Watchdog plc 2 ok
OUT M_Hardw_Watchdogs_Plc1_Plc2_OK  ; Merker Hardware Watchdogs Plc 1 & Plc 2 OK

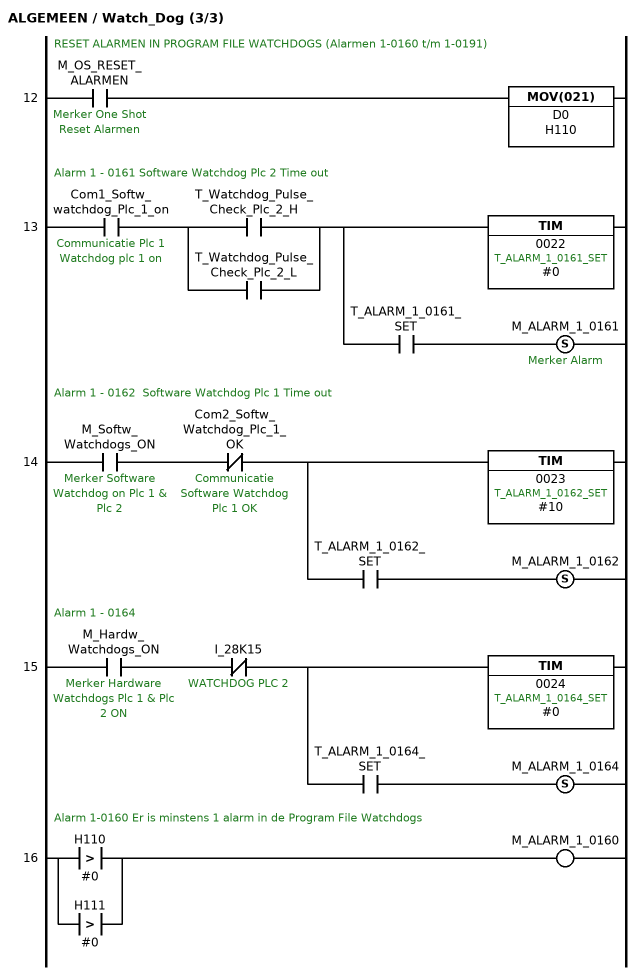
; rung 12: RESET ALARMEN IN PROGRAM FILE WATCHDOGS (Alarmen 1-0160 t/m 1-0191)
LD M_OS_RESET_ALARMEN  ; Merker One Shot Reset Alarmen
MOV(021) D0 H110
; rung 13: Alarm 1 - 0161 Software Watchdog Plc 2 Time out
LD Com1_Softw_watchdog_Plc_1_on  ; Communicatie Plc 1 Watchdog plc 1 on
LD T_Watchdog_Pulse_Check_Plc_2_H
OR T_Watchdog_Pulse_Check_Plc_2_L
ANDLD
TIM 0022 #0  ; T_ALARM_1_0161_SET
AND T_ALARM_1_0161_SET
SET M_ALARM_1_0161  ; Merker Alarm
; rung 14: Alarm 1 - 0162  Software Watchdog Plc 1 Time out
LD M_Softw_Watchdogs_ON  ; Merker Software Watchdog on Plc 1 & Plc 2
ANDNOT Com2_Softw_Watchdog_Plc_1_OK  ; Communicatie Software Watchdog Plc 1 OK
TIM 0023 #10  ; T_ALARM_1_0162_SET
AND T_ALARM_1_0162_SET
SET M_ALARM_1_0162
; rung 15: Alarm 1 - 0164
LD M_Hardw_Watchdogs_ON  ; Merker Hardware Watchdogs Plc 1 & Plc 2 ON
ANDNOT I_28K15  ; WATCHDOG PLC 2
TIM 0024 #0  ; T_ALARM_1_0164_SET
AND T_ALARM_1_0164_SET
SET M_ALARM_1_0164
; rung 16: Alarm 1-0160 Er is minstens 1 alarm in de Program File Watchdogs
LD>(320) H110 #0
OR>(320) H111 #0
OUT M_ALARM_1_0160

### Section E_Stops

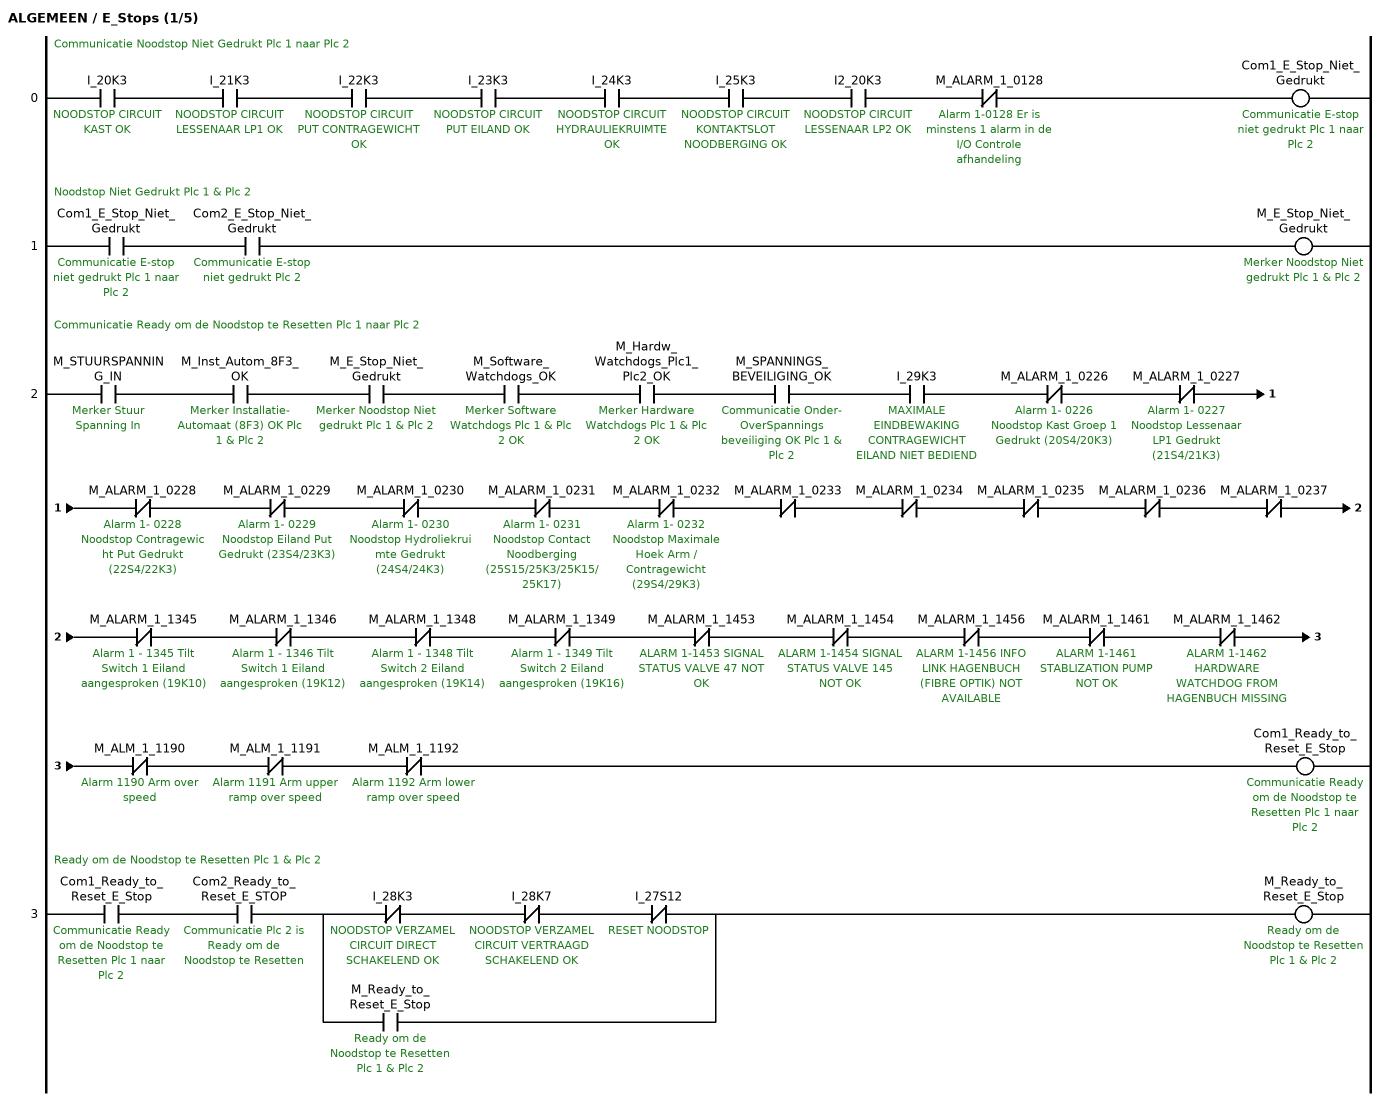
; rung 0: Communicatie Noodstop Niet Gedrukt Plc 1 naar Plc 2
LD I_20K3  ; NOODSTOP CIRCUIT KAST OK
AND I_21K3  ; NOODSTOP CIRCUIT LESSENAAR LP1 OK
AND I_22K3  ; NOODSTOP CIRCUIT PUT CONTRAGEWICHT OK
AND I_23K3  ; NOODSTOP CIRCUIT PUT EILAND OK
AND I_24K3  ; NOODSTOP CIRCUIT HYDRAULIEKRUIMTE OK
AND I_25K3  ; NOODSTOP CIRCUIT KONTAKTSLOT NOODBERGING OK
AND I2_20K3  ; NOODSTOP CIRCUIT LESSENAAR LP2 OK
ANDNOT M_ALARM_1_0128  ; Alarm 1-0128 Er is minstens 1 alarm in de I/O Controle afhandeling
OUT Com1_E_Stop_Niet_Gedrukt  ; Communicatie E-stop niet gedrukt Plc 1 naar Plc 2
; rung 1: Noodstop Niet Gedrukt Plc 1 & Plc 2
LD Com1_E_Stop_Niet_Gedrukt  ; Communicatie E-stop niet gedrukt Plc 1 naar Plc 2
AND Com2_E_Stop_Niet_Gedrukt  ; Communicatie E-stop niet gedrukt Plc 2
OUT M_E_Stop_Niet_Gedrukt  ; Merker Noodstop Niet gedrukt Plc 1 & Plc 2
; rung 2: Communicatie Ready om de Noodstop te Resetten Plc 1 naar Plc 2
LD M_STUURSPANNING_IN  ; Merker Stuur Spanning In
AND M_Inst_Autom_8F3_OK  ; Merker Installatie-Automaat (8F3) OK Plc 1 & Plc 2
AND M_E_Stop_Niet_Gedrukt  ; Merker Noodstop Niet gedrukt Plc 1 & Plc 2
AND M_Software_Watchdogs_OK  ; Merker Software Watchdogs Plc 1 & Plc 2 OK
AND M_Hardw_Watchdogs_Plc1_Plc2_OK  ; Merker Hardware Watchdogs Plc 1 & Plc 2 OK
AND M_SPANNINGS_BEVEILIGING_OK  ; Communicatie Onder- OverSpannings beveiliging OK Plc 1 & Plc 2
AND I_29K3  ; MAXIMALE EINDBEWAKING CONTRAGEWICHT EILAND NIET BEDIEND
ANDNOT M_ALARM_1_0226  ; Alarm 1- 0226 Noodstop Kast Groep 1 Gedrukt (20S4/20K3)
ANDNOT M_ALARM_1_0227  ; Alarm 1- 0227 Noodstop Lessenaar LP1 Gedrukt (21S4/21K3)
ANDNOT M_ALARM_1_0228  ; Alarm 1- 0228 Noodstop Contragewicht Put Gedrukt (22S4/22K3)
ANDNOT M_ALARM_1_0229  ; Alarm 1- 0229 Noodstop Eiland Put Gedrukt (23S4/23K3)
ANDNOT M_ALARM_1_0230  ; Alarm 1- 0230 Noodstop Hydroliekruimte Gedrukt (24S4/24K3)
ANDNOT M_ALARM_1_0231  ; Alarm 1- 0231 Noodstop Contact Noodberging (25S15/25K3/25K15/25K17)
ANDNOT M_ALARM_1_0232  ; Alarm 1- 0232 Noodstop Maximale Hoek Arm / Contragewicht  (29S4/29K3)
ANDNOT M_ALARM_1_0233
ANDNOT M_ALARM_1_0234
ANDNOT M_ALARM_1_0235
ANDNOT M_ALARM_1_0236
ANDNOT M_ALARM_1_0237
ANDNOT M_ALARM_1_1345  ; Alarm 1 - 1345 Tilt Switch 1 Eiland aangesproken (19K10)
ANDNOT M_ALARM_1_1346  ; Alarm 1 - 1346 Tilt Switch 1 Eiland aangesproken (19K12)
ANDNOT M_ALARM_1_1348  ; Alarm 1 - 1348 Tilt Switch 2 Eiland aangesproken (19K14)
ANDNOT M_ALARM_1_1349  ; Alarm 1 - 1349 Tilt Switch 2 Eiland aangesproken (19K16)
ANDNOT M_ALARM_1_1453  ; ALARM 1-1453 SIGNAL STATUS VALVE 47 NOT OK
ANDNOT M_ALARM_1_1454  ; ALARM 1-1454 SIGNAL STATUS VALVE 145 NOT OK
ANDNOT M_ALARM_1_1456  ; ALARM 1-1456 INFO LINK HAGENBUCH (FIBRE OPTIK) NOT AVAILABLE
ANDNOT M_ALARM_1_1461  ; ALARM 1-1461 STABLIZATION PUMP NOT OK
ANDNOT M_ALARM_1_1462  ; ALARM 1-1462 HARDWARE WATCHDOG FROM HAGENBUCH MISSING
ANDNOT M_ALM_1_1190  ; Alarm 1190 Arm over speed
ANDNOT M_ALM_1_1191  ; Alarm 1191 Arm upper ramp over speed
ANDNOT M_ALM_1_1192  ; Alarm 1192 Arm lower ramp over speed
OUT Com1_Ready_to_Reset_E_Stop  ; Communicatie Ready om de Noodstop te Resetten Plc 1 naar Plc 2
; rung 3: Ready om de Noodstop te Resetten Plc 1 & Plc 2
LD Com1_Ready_to_Reset_E_Stop  ; Communicatie Ready om de Noodstop te Resetten Plc 1 naar Plc 2
AND Com2_Ready_to_Reset_E_STOP  ; Communicatie Plc 2 is Ready om de Noodstop te Resetten
LDNOT I_28K3  ; NOODSTOP VERZAMEL CIRCUIT DIRECT SCHAKELEND OK
ANDNOT I_28K7  ; NOODSTOP VERZAMEL CIRCUIT VERTRAAGD SCHAKELEND OK
ANDNOT I_27S12  ; RESET NOODSTOP
OR M_Ready_to_Reset_E_Stop  ; Ready om de Noodstop te Resetten Plc 1 & Plc 2
ANDLD
OUT M_Ready_to_Reset_E_Stop  ; Ready om de Noodstop te Resetten Plc 1 & Plc 2

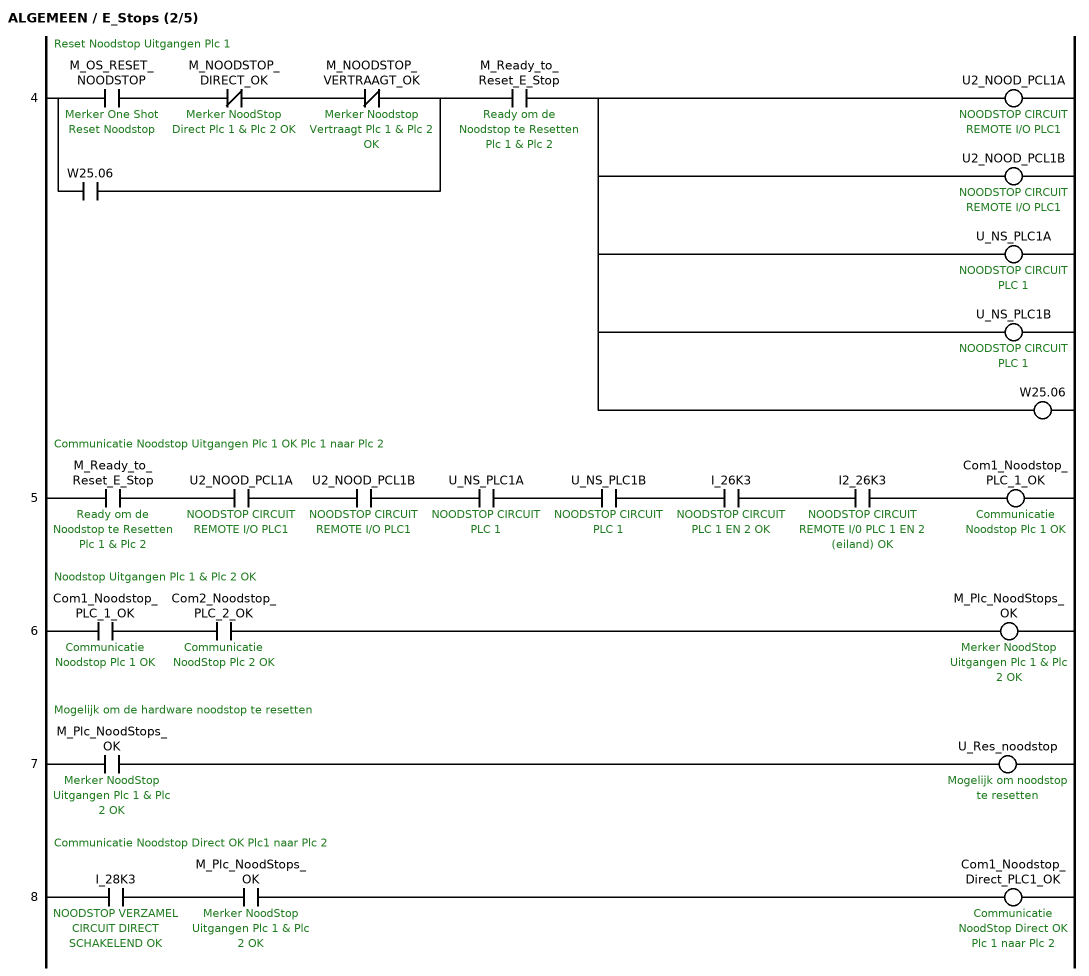
; rung 4: Reset Noodstop Uitgangen Plc 1
LD M_OS_RESET_NOODSTOP  ; Merker One Shot  Reset Noodstop
ANDNOT M_NOODSTOP_DIRECT_OK  ; Merker NoodStop Direct Plc 1 & Plc 2 OK
ANDNOT M_NOODSTOP_VERTRAAGT_OK  ; Merker Noodstop Vertraagt Plc 1 & Plc 2 OK
OR W25.06
AND M_Ready_to_Reset_E_Stop  ; Ready om de Noodstop te Resetten Plc 1 & Plc 2
OUT U2_NOOD_PCL1A  ; NOODSTOP CIRCUIT REMOTE I/O PLC1
OUT U2_NOOD_PCL1B  ; NOODSTOP CIRCUIT REMOTE I/O PLC1
OUT U_NS_PLC1A  ; NOODSTOP CIRCUIT PLC 1
OUT U_NS_PLC1B  ; NOODSTOP CIRCUIT PLC 1
OUT W25.06
; rung 5: Communicatie Noodstop Uitgangen Plc 1 OK Plc 1 naar Plc 2
LD M_Ready_to_Reset_E_Stop  ; Ready om de Noodstop te Resetten Plc 1 & Plc 2
AND U2_NOOD_PCL1A  ; NOODSTOP CIRCUIT REMOTE I/O PLC1
AND U2_NOOD_PCL1B  ; NOODSTOP CIRCUIT REMOTE I/O PLC1
AND U_NS_PLC1A  ; NOODSTOP CIRCUIT PLC 1
AND U_NS_PLC1B  ; NOODSTOP CIRCUIT PLC 1
AND I_26K3  ; NOODSTOP CIRCUIT PLC 1 EN 2 OK
AND I2_26K3  ; NOODSTOP CIRCUIT REMOTE I/0 PLC 1 EN 2 (eiland) OK
OUT Com1_Noodstop_PLC_1_OK  ; Communicatie Noodstop Plc 1 OK
; rung 6: Noodstop Uitgangen Plc 1 & Plc 2 OK
LD Com1_Noodstop_PLC_1_OK  ; Communicatie Noodstop Plc 1 OK
AND Com2_Noodstop_PLC_2_OK  ; Communicatie NoodStop Plc 2 OK
OUT M_Plc_NoodStops_OK  ; Merker NoodStop Uitgangen Plc 1 & Plc 2 OK
; rung 7: Mogelijk om de hardware noodstop te resetten
LD M_Plc_NoodStops_OK  ; Merker NoodStop Uitgangen Plc 1 & Plc 2 OK
OUT U_Res_noodstop  ; Mogelijk om noodstop te resetten
; rung 8: Communicatie Noodstop Direct OK Plc1 naar Plc 2
LD I_28K3  ; NOODSTOP VERZAMEL CIRCUIT DIRECT SCHAKELEND OK
AND M_Plc_NoodStops_OK  ; Merker NoodStop Uitgangen Plc 1 & Plc 2 OK
OUT Com1_Noodstop_Direct_PLC1_OK  ; Communicatie NoodStop Direct OK Plc 1 naar Plc 2

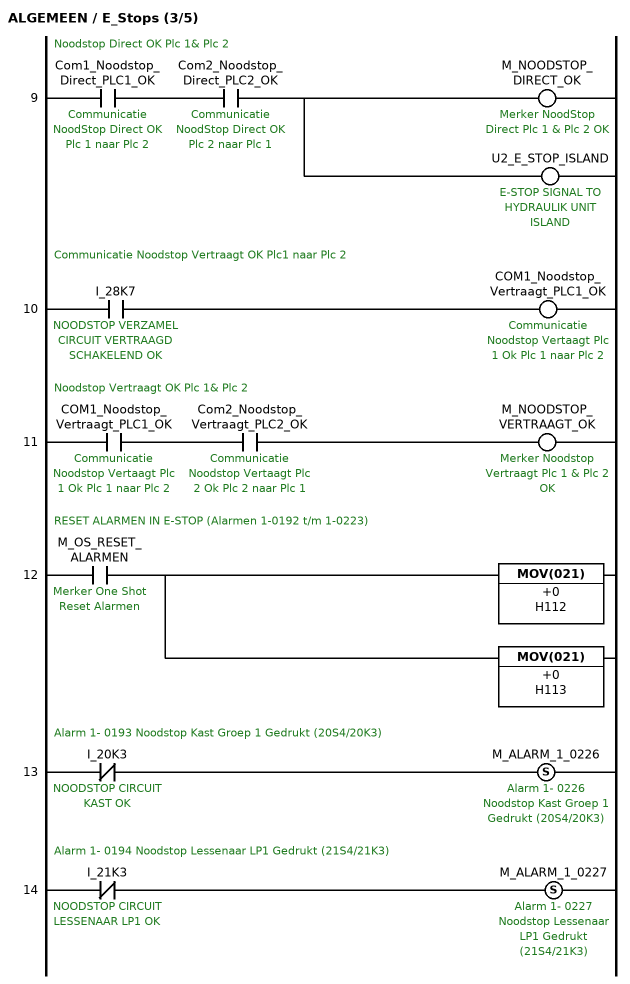
; rung 9: Noodstop Direct OK Plc 1& Plc 2
LD Com1_Noodstop_Direct_PLC1_OK  ; Communicatie NoodStop Direct OK Plc 1 naar Plc 2
AND Com2_Noodstop_Direct_PLC2_OK  ; Communicatie NoodStop Direct OK Plc 2 naar Plc 1
OUT M_NOODSTOP_DIRECT_OK  ; Merker NoodStop Direct Plc 1 & Plc 2 OK
OUT U2_E_STOP_ISLAND  ; E-STOP SIGNAL TO HYDRAULIK UNIT ISLAND
; rung 10: Communicatie Noodstop Vertraagt OK Plc1 naar Plc 2
LD I_28K7  ; NOODSTOP VERZAMEL CIRCUIT VERTRAAGD SCHAKELEND OK
OUT COM1_Noodstop_Vertraagt_PLC1_OK  ; Communicatie Noodstop Vertaagt Plc 1 Ok Plc 1 naar Plc 2
; rung 11: Noodstop Vertraagt OK Plc 1& Plc 2
LD COM1_Noodstop_Vertraagt_PLC1_OK  ; Communicatie Noodstop Vertaagt Plc 1 Ok Plc 1 naar Plc 2
AND Com2_Noodstop_Vertraagt_PLC2_OK  ; Communicatie Noodstop Vertaagt Plc 2 Ok Plc 2 naar Plc 1
OUT M_NOODSTOP_VERTRAAGT_OK  ; Merker Noodstop Vertraagt Plc 1 & Plc 2 OK
; rung 12: RESET ALARMEN IN E-STOP (Alarmen 1-0192 t/m 1-0223)
LD M_OS_RESET_ALARMEN  ; Merker One Shot Reset Alarmen
MOV(021) +0 H112
MOV(021) +0 H113
; rung 13: Alarm 1- 0193 Noodstop Kast Groep 1 Gedrukt (20S4/20K3)
LDNOT I_20K3  ; NOODSTOP CIRCUIT KAST OK
SET M_ALARM_1_0226  ; Alarm 1- 0226 Noodstop Kast Groep 1 Gedrukt (20S4/20K3)
; rung 14: Alarm 1- 0194 Noodstop Lessenaar LP1 Gedrukt (21S4/21K3)
LDNOT I_21K3  ; NOODSTOP CIRCUIT LESSENAAR LP1 OK
SET M_ALARM_1_0227  ; Alarm 1- 0227 Noodstop Lessenaar LP1 Gedrukt (21S4/21K3)

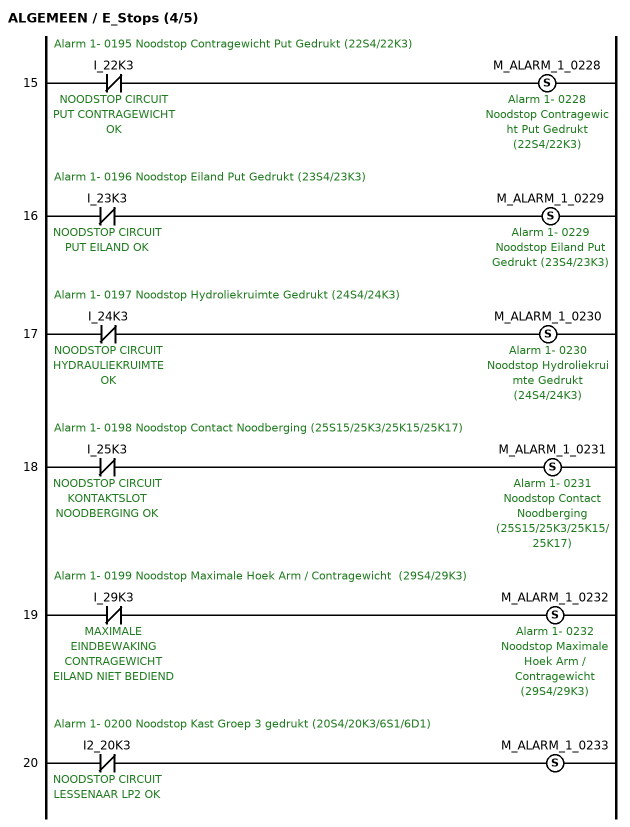
; rung 15: Alarm 1- 0195 Noodstop Contragewicht Put Gedrukt (22S4/22K3)
LDNOT I_22K3  ; NOODSTOP CIRCUIT PUT CONTRAGEWICHT OK
SET M_ALARM_1_0228  ; Alarm 1- 0228 Noodstop Contragewicht Put Gedrukt (22S4/22K3)
; rung 16: Alarm 1- 0196 Noodstop Eiland Put Gedrukt (23S4/23K3)
LDNOT I_23K3  ; NOODSTOP CIRCUIT PUT EILAND OK
SET M_ALARM_1_0229  ; Alarm 1- 0229 Noodstop Eiland Put Gedrukt (23S4/23K3)
; rung 17: Alarm 1- 0197 Noodstop Hydroliekruimte Gedrukt (24S4/24K3)
LDNOT I_24K3  ; NOODSTOP CIRCUIT HYDRAULIEKRUIMTE OK
SET M_ALARM_1_0230  ; Alarm 1- 0230 Noodstop Hydroliekruimte Gedrukt (24S4/24K3)
; rung 18: Alarm 1- 0198 Noodstop Contact Noodberging (25S15/25K3/25K15/25K17)
LDNOT I_25K3  ; NOODSTOP CIRCUIT KONTAKTSLOT NOODBERGING OK
SET M_ALARM_1_0231  ; Alarm 1- 0231 Noodstop Contact Noodberging (25S15/25K3/25K15/25K17)
; rung 19: Alarm 1- 0199 Noodstop Maximale Hoek Arm / Contragewicht  (29S4/29K3)
LDNOT I_29K3  ; MAXIMALE EINDBEWAKING CONTRAGEWICHT EILAND NIET BEDIEND
SET M_ALARM_1_0232  ; Alarm 1- 0232 Noodstop Maximale Hoek Arm / Contragewicht  (29S4/29K3)
; rung 20: Alarm 1- 0200 Noodstop Kast Groep 3 gedrukt (20S4/20K3/6S1/6D1)
LDNOT I2_20K3  ; NOODSTOP CIRCUIT LESSENAAR LP2 OK
SET M_ALARM_1_0233

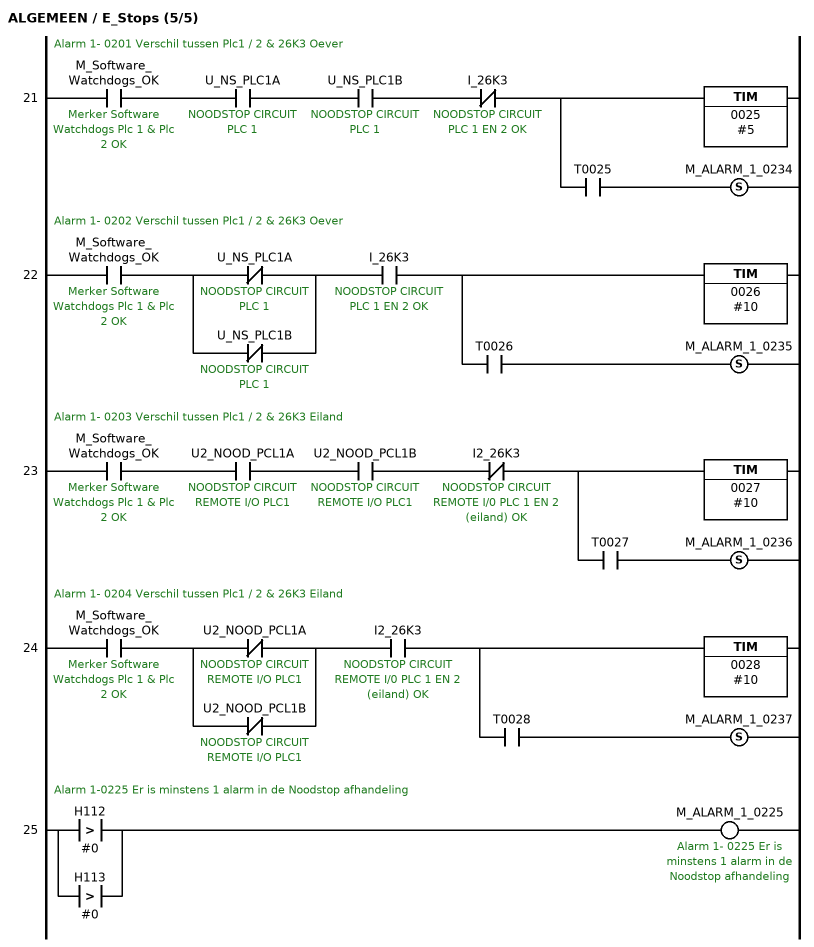
; rung 21: Alarm 1- 0201 Verschil tussen Plc1 / 2 & 26K3 Oever
LD M_Software_Watchdogs_OK  ; Merker Software Watchdogs Plc 1 & Plc 2 OK
AND U_NS_PLC1A  ; NOODSTOP CIRCUIT PLC 1
AND U_NS_PLC1B  ; NOODSTOP CIRCUIT PLC 1
ANDNOT I_26K3  ; NOODSTOP CIRCUIT PLC 1 EN 2 OK
TIM 0025 #5
AND T0025
SET M_ALARM_1_0234
; rung 22: Alarm 1- 0202 Verschil tussen Plc1 / 2 & 26K3 Oever
LD M_Software_Watchdogs_OK  ; Merker Software Watchdogs Plc 1 & Plc 2 OK
LDNOT U_NS_PLC1A  ; NOODSTOP CIRCUIT PLC 1
ORNOT U_NS_PLC1B  ; NOODSTOP CIRCUIT PLC 1
ANDLD
AND I_26K3  ; NOODSTOP CIRCUIT PLC 1 EN 2 OK
TIM 0026 #10
AND T0026
SET M_ALARM_1_0235
; rung 23: Alarm 1- 0203 Verschil tussen Plc1 / 2 & 26K3 Eiland
LD M_Software_Watchdogs_OK  ; Merker Software Watchdogs Plc 1 & Plc 2 OK
AND U2_NOOD_PCL1A  ; NOODSTOP CIRCUIT REMOTE I/O PLC1
AND U2_NOOD_PCL1B  ; NOODSTOP CIRCUIT REMOTE I/O PLC1
ANDNOT I2_26K3  ; NOODSTOP CIRCUIT REMOTE I/0 PLC 1 EN 2 (eiland) OK
TIM 0027 #10
AND T0027
SET M_ALARM_1_0236
; rung 24: Alarm 1- 0204 Verschil tussen Plc1 / 2 & 26K3 Eiland
LD M_Software_Watchdogs_OK  ; Merker Software Watchdogs Plc 1 & Plc 2 OK
LDNOT U2_NOOD_PCL1A  ; NOODSTOP CIRCUIT REMOTE I/O PLC1
ORNOT U2_NOOD_PCL1B  ; NOODSTOP CIRCUIT REMOTE I/O PLC1
ANDLD
AND I2_26K3  ; NOODSTOP CIRCUIT REMOTE I/0 PLC 1 EN 2 (eiland) OK
TIM 0028 #10
AND T0028
SET M_ALARM_1_0237
; rung 25: Alarm 1-0225 Er is minstens 1 alarm in de Noodstop afhandeling
LD>(320) H112 #0
OR>(320) H113 #0
OUT M_ALARM_1_0225  ; Alarm 1- 0225 Er is minstens 1 alarm in de Noodstop afhandeling

### Section Configure_I_O

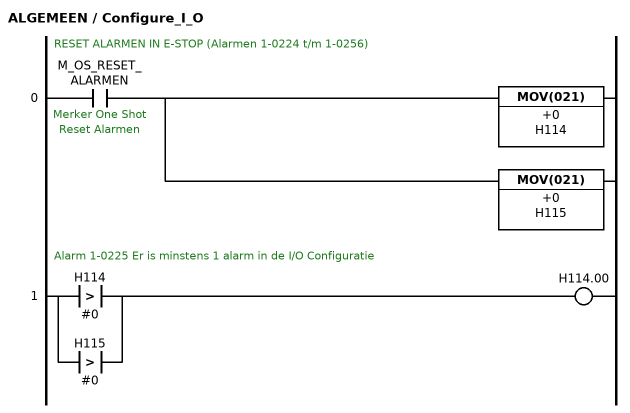
; rung 0: RESET ALARMEN IN E-STOP (Alarmen 1-0224 t/m 1-0256)
LD M_OS_RESET_ALARMEN  ; Merker One Shot Reset Alarmen
MOV(021) +0 H114
MOV(021) +0 H115
; rung 1: Alarm 1-0225 Er is minstens 1 alarm in de I/O Configuratie
LD>(320) H114 #0
OR>(320) H115 #0
OUT H114.00

### Section Wind_Meeting
; rung 0: De Windmeting word ingelezen in Plc 2

